Staubli VAL3: PickPlace.pgx

program PickPlace()
begin


  while true

    wait(bNewData)

    if bPick
      call pick(nX,nY)
    else
      call place(nX,nY)
    endIf


    bNewData = false
    bReady = true



  endWhile

end
